Omron CX-Programmer project NewProject (CX-Programmer 9.75)

# PLC BottleFillingAutomated: CP1E N30

## Global symbols (name address type ; comment)
T000 BOOL  ; T0
T001 BOOL  ; T1
T002 BOOL  ; T2
T003 BOOL  ; T3
T004 BOOL  ; T4
T005 BOOL  ; T5

## Program NewProgram1 (cyclic task 0)
Local symbols
CapingMotor 100.03 BOOL  ; 100.03
ConvyerMotor 100.01 BOOL  ; 100.01
LabelMotor 100.04 BOOL  ; 100.04
MainSupply 100.00 BOOL  ; 100.00
Sensor 0.02 BOOL  ; 0.02
Start 0.00 BOOL  ; 0.00
Stop 0.01 BOOL  ; 0.01
Valve 100.02 BOOL  ; 100.02

### Section Section1

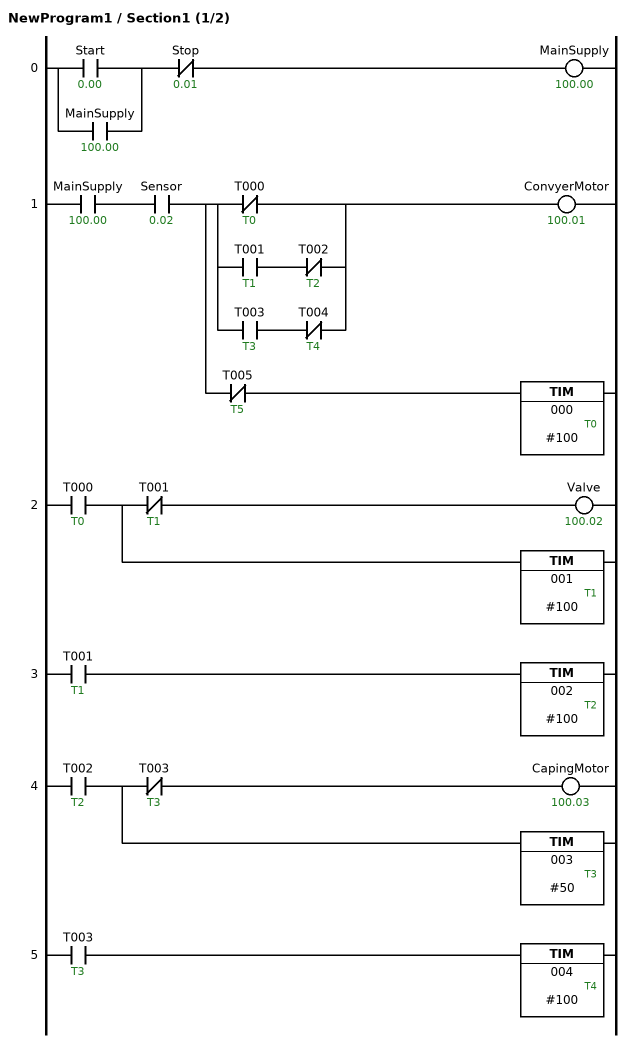
; rung 0
LD Start  ; 0.00
OR MainSupply  ; 100.00
ANDNOT Stop  ; 0.01
OUT MainSupply  ; 100.00
; rung 1
LD MainSupply  ; 100.00
AND Sensor  ; 0.02
OUT TR0
LDNOT T000  ; T0
LD T001  ; T1
ANDNOT T002  ; T2
ORLD
LD T003  ; T3
ANDNOT T004  ; T4
ORLD
ANDLD
OUT ConvyerMotor  ; 100.01
LD TR0
ANDNOT T005  ; T5
TIM 000 #100  ; T0
; rung 2
LD T000  ; T0
OUT TR0
ANDNOT T001  ; T1
OUT Valve  ; 100.02
LD TR0
TIM 001 #100  ; T1
; rung 3
LD T001  ; T1
TIM 002 #100  ; T2
; rung 4
LD T002  ; T2
OUT TR0
ANDNOT T003  ; T3
OUT CapingMotor  ; 100.03
LD TR0
TIM 003 #50  ; T3
; rung 5
LD T003  ; T3
TIM 004 #100  ; T4

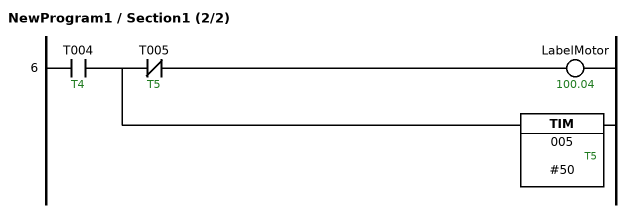
; rung 6
LD T004  ; T4
OUT TR0
ANDNOT T005  ; T5
OUT LabelMotor  ; 100.04
LD TR0
TIM 005 #50  ; T5

### Section END
; rung 0
END(001)